TYPE ST_RGBW_Steuerung :
STRUCT
	Betrieb			: BOOL;
	Farbcode	: STRING;
END_STRUCT
END_TYPE

(* stored: Version 1.1.0.1, ProductVersion 3.1.4024.10
   DUT ST_RGBW_Steuerung: Id {1f51ad7e-988c-4471-a02b-1b8075025710} *)
